FUNCTION_BLOCK HAL

							  
//--{attribute 'TcLinkTo' := 'TIID^Master (EtherCAT)^Term 1 (EK1200)^Term 7 (EL1008)^Channel 1^Input'}
//--     bVarIn2    AT%I*  : BOOL;  // linked via attribute 
	
// kan ook worden gebruikt om te verwijzen naar een andere PLC.
// Dit zou met name handig kunnen zijn wanneer er geschakel moet worden tussen Device Hardware en het simulatie projedt.
// Dan worden de linkings automatische gegenereerd, en hoeft dit dus niet meer handmatig te worden gedaan. |Veel tijd winst en kan op minder  fouiten.

//-{attribute 'TcLinkTo' := 'TIID^Master (EtherCAT)^Term 1 (EK1200)^Term 9 (EL1809)^Channel 1^Input'}
//-MAIN.GVL_Modules.g_emDockingInterface.s_cmDockingClampsUpper.I_bStaValveIsOn AT%I* : BOOL;


//--GVL_Modules.g_emDockingInterface.s_cmDockingClampsUpper.I_bStaValveIsOn := MAIN.GVL_Modules_g_emDockingInterface_s_cmDockingClampsUpper_I_bStaValveIsOn;

//--GVL_Modules.g_emUtilities.s_diSafetyOk.I_bStaInput := MAIN.GVL_Modules_g_emUtilities_s_diSafetyOk_I_bStaInput;
//--GVL_Modules.g_emUtilities.s_di24VdcOk.I_bStaInput := MAIN.GVL_Modules_g_emUtilities_s_di24VdcOk_I_bStaInput;
//--GVL_Modules.g_emUtilities.s_diAirPressureOk.I_bStaInput := MAIN.GVL_Modules_g_emUtilities_s_diAirPressureOk_I_bStaInput;

END_FUNCTION_BLOCK

(* stored: Version 1.1.0.1, ProductVersion 3.1.4024.12
   POU HAL: Id {3a9bd6e1-4674-4645-a5d3-1835b5ad1e40}, SpecialFunc None *)
